FUNCTION_BLOCK ConveyorAdvanced_2 (* Basic Function Block Type *)
  (* Standard: 61499-2 *)
  (* Version 0.0, 9/24/2018, dmidro, nxtControl GmbH, Template *)
  PACKAGE Main;
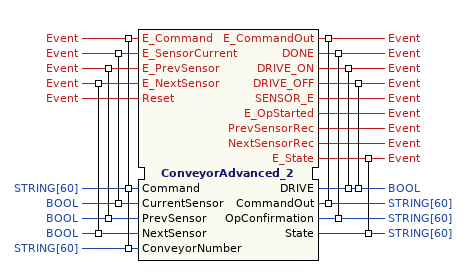
  EVENT_INPUT
    E_Command WITH Command, ConveyorNumber;
    E_SensorCurrent WITH CurrentSensor;
    E_PrevSensor WITH PrevSensor;
    E_NextSensor WITH NextSensor;
    Reset;
  END_EVENT
  EVENT_OUTPUT
    E_CommandOut WITH CommandOut;
    DONE WITH OpConfirmation; (* Execution Confirmation *)
    DRIVE_ON WITH DRIVE;
    DRIVE_OFF WITH DRIVE;
    SENSOR_E;
    E_OpStarted;
    PrevSensorRec;
    NextSensorRec;
    E_State WITH State;
  END_EVENT
  VAR_INPUT
    Command : STRING[60];
    CurrentSensor : BOOL; {SET_ATTRIBUTE(Runtime.OPCUA.Access, 2)} {SET_ATTRIBUTE(Runtime.OPCUA.WriteTrigger, SENSOR)}
    PrevSensor : BOOL;
    NextSensor : BOOL;
    ConveyorNumber : STRING[60];
  END_VAR
  VAR_OUTPUT
    DRIVE : BOOL; {SET_ATTRIBUTE(Runtime.OPCUA.Access, 2)}
    CommandOut : STRING[60];
    OpConfirmation : STRING[60];
    State : STRING[60];
  END_VAR
  VAR
    C : STRING[60];
    P : STRING[60];
    D : STRING[60];
    commandCheck : STRING[60];
    TriggerDelivery : BOOL;
    TriggerConveyor : BOOL;
    TriggerWait : BOOL;
    Suspend : BOOL;
    C_INT : DINT;
    D_INT : DINT;
    P_INT : DINT;
  END_VAR
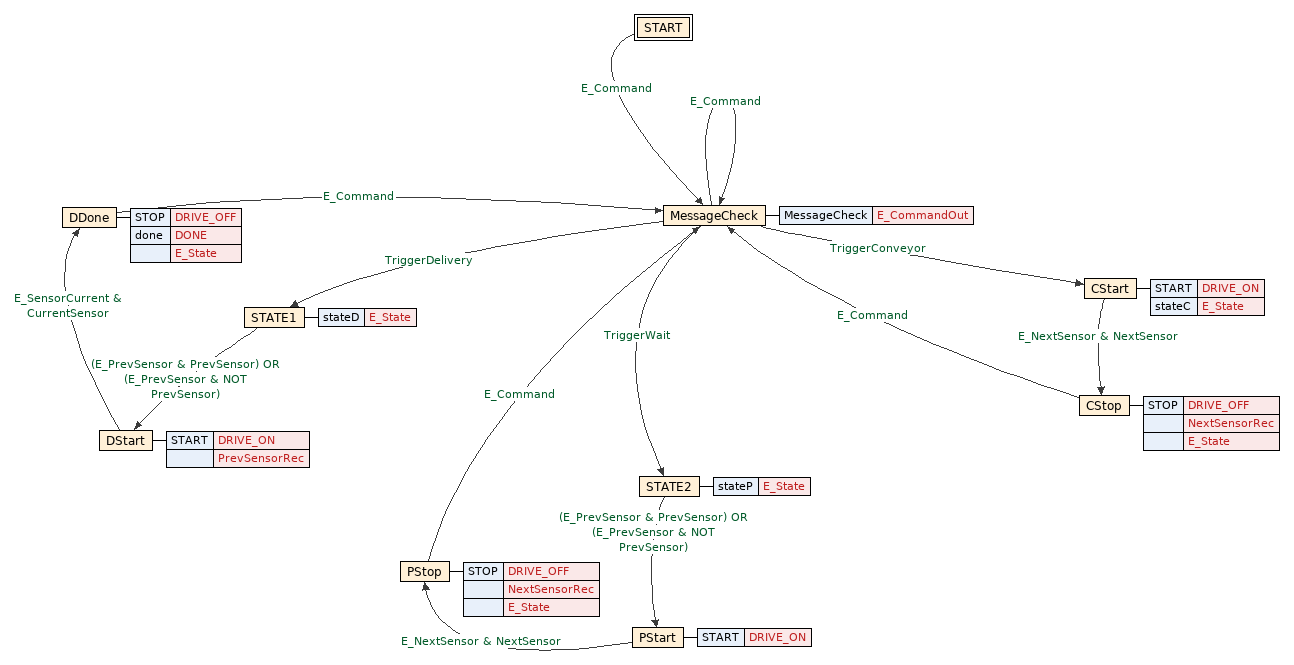
  EC_STATES
    START; (* Initial State *)
    MessageCheck : MessageCheck -> E_CommandOut;
    DStart : START -> DRIVE_ON, -> PrevSensorRec;
    CStart : START -> DRIVE_ON, stateC -> E_State;
    DDone : STOP -> DRIVE_OFF, done -> DONE, -> E_State;
    CStop : STOP -> DRIVE_OFF, -> NextSensorRec, -> E_State;
    PStart : START -> DRIVE_ON;
    PStop : STOP -> DRIVE_OFF, -> NextSensorRec, -> E_State;
    STATE1 : stateD -> E_State;
    STATE2 : stateP -> E_State;
  END_STATES
  EC_TRANSITIONS
    START TO MessageCheck := E_Command;
    MessageCheck TO STATE1 := TriggerDelivery;
    MessageCheck TO STATE2 := TriggerWait;
    MessageCheck TO CStart := TriggerConveyor;
    DStart TO DDone := E_SensorCurrent & CurrentSensor;
    DDone TO MessageCheck := E_Command;
    CStart TO CStop := E_NextSensor & NextSensor;
    CStop TO MessageCheck := E_Command;
    PStop TO MessageCheck := E_Command;
    PStart TO PStop := E_NextSensor & NextSensor;
    STATE1 TO DStart := (E_PrevSensor & PrevSensor) OR (E_PrevSensor & NOT PrevSensor);
    MessageCheck TO MessageCheck := E_Command;
    STATE2 TO PStart := (E_PrevSensor & PrevSensor) OR (E_PrevSensor & NOT PrevSensor);
  END_TRANSITIONS
  ALGORITHM INIT IN ST: (* Initialization algorithm *)
;
  END_ALGORITHM
  ALGORITHM MessageCheck IN ST: (* Normally executed algorithm *)
// commandCheck := LEFT(Command,2);
C := CONCAT('C',ConveyorNumber);
P := CONCAT('P',ConveyorNumber);
D := CONCAT('D',ConveyorNumber);

C_INT := FIND(Command,C);
P_INT := FIND(Command,P);
D_INT := FIND(Command,D);

IF C_INT = 1 THEN
	TriggerConveyor := TRUE;
	CommandOut := DELETE(Command,3,1);
ELSIF P_INT = 1 THEN
	TriggerWait := TRUE;
	CommandOut := DELETE(Command,3,1);
ELSIF D_INT = 1 THEN
	TriggerDelivery := TRUE;
	CommandOut := DELETE(Command,3,1);

ELSE
	Suspend := TRUE;
	CommandOut := Command;
END_IF;
  END_ALGORITHM
  ALGORITHM START IN ST:
DRIVE := TRUE;
  END_ALGORITHM
  ALGORITHM STOP IN ST:
DRIVE := FALSE;

TriggerConveyor := FALSE;
TriggerDelivery := FALSE;
TriggerWait := FALSE;
State := '';
  END_ALGORITHM
  ALGORITHM done IN ST:
OpConfirmation := CONCAT('C',ConveyorNumber,'_DONE');
  END_ALGORITHM
  ALGORITHM Suspend IN ST:
Suspend := FALSE;
  END_ALGORITHM
  ALGORITHM stateD IN ST:
State := CONCAT('D',ConveyorNumber);
  END_ALGORITHM
  ALGORITHM stateP IN ST:
State := CONCAT('P',ConveyorNumber);
  END_ALGORITHM
  ALGORITHM stateC IN ST:
State := CONCAT('C',ConveyorNumber);
  END_ALGORITHM
END_FUNCTION_BLOCK
